(* Logix 5000 project; controller plcgr3 vendor 1 type 14 code 89 rev 20.19; software revision 20.05 *)

TASK MainTask (continuous, watchdog 500 ms) : MainProgram

MODULES
   Controller : vendor 1 type 14 code 89 (CompactLogixL23E_QBFC1_Controller 0, rev 20.19)
      LocalENB : vendor 1 type 12 code 191 (CompactLogixL23E_QBFC1_Ethernet 1, Ethernet 192.168.10.8, rev 20.11)
      Local : CompactBus (CompactVirtualAdapter 3, rev 20.11)
         Discrete_Inputs : vendor 1 type 7 code 320 (Compact 1, rev 3.1, Input RPI 20 ms)
         Analog_IO : vendor 1 type 10 code 120 (Compact 3, rev 1.1, Output RPI 80 ms)
         Counters : vendor 1 type 109 code 70 (Compact 4, rev 1.1, Output RPI 20 ms)
         Discrete_Outputs : vendor 1 type 7 code 322 (Compact 2, rev 3.1, Output RPI 20 ms)
         scanner : vendor 1 type 12 code 105 (Compact 5, rev 3.1, Output RPI 20 ms)
END_MODULES

PROGRAM MainProgram   (* main routine MainRoutine *)
VAR
   Comando : ALIAS FOR Local:5:O.Data[0];
   comando_aux : DINT := 39520;
   motor : BOOL;
   start : ALIAS FOR Local:1:I.Data.0;
   start_HMi : BOOL;
   stop : ALIAS FOR Local:1:I.Data.1;
   stop_HMI : BOOL;
   Velocidad : DINT := 12000;
   velocidad_aux : DINT := 12000;
   velocidad_aux2 : DINT := 786432000;
END_VAR

ROUTINE MainRoutine   (* ladder *)
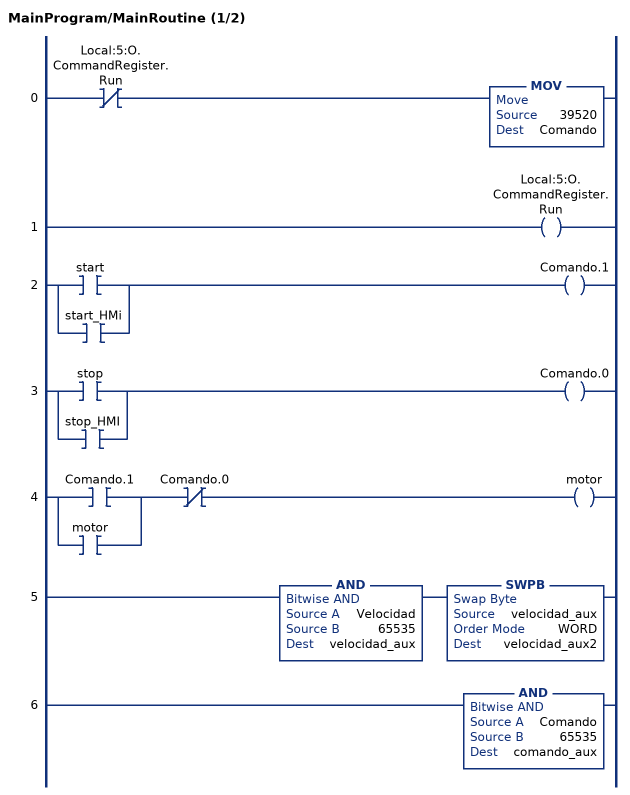
   0: XIO(Local:5:O.CommandRegister.Run)MOV(39520,Comando);
   1: OTE(Local:5:O.CommandRegister.Run);
   2: [XIC(start) ,XIC(start_HMi) ]OTE(Comando.1);
   3: [XIC(stop) ,XIC(stop_HMI) ]OTE(Comando.0);
   4: [XIC(Comando.1) ,XIC(motor) ]XIO(Comando.0)OTE(motor);
   5: AND(Velocidad,65535,velocidad_aux)SWPB(velocidad_aux,WORD,velocidad_aux2);
   6: AND(Comando,65535,comando_aux);
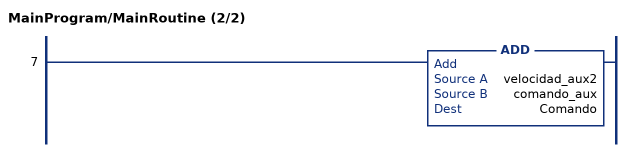
   7: ADD(velocidad_aux2,comando_aux,Comando);
END_ROUTINE
END_PROGRAM
